(* IEC 61131-3 sources: CodigoPPC/FB da IHM, 6 files *)

(* ---- FC_EpochToString.st ---- *)
// ════════════════════════════════════════════════════════════════════
// FC_EpochToString — Converte UDINT epoch UTC para string legível
// ════════════════════════════════════════════════════════════════════
// Formato: 'DD/MM HH:MM:SS'
// Simplificação: usa SysTimeRtcConvertUtcToLocal + formatação manual
// Se tTimestamp = 0, retorna '-- sem RTC --'
// ════════════════════════════════════════════════════════════════════
FUNCTION FC_EpochToString : STRING(20)
VAR_INPUT
    tEpoch : UDINT;
END_VAR
VAR
    dtLocal     : DT;
    sTemp       : STRING(20);
    nDay        : UINT;
    nMonth      : UINT;
    nHour       : UINT;
    nMin        : UINT;
    nSec        : UINT;
END_VAR

    IF tEpoch = 0 THEN
        FC_EpochToString := '-- sem RTC --';
        RETURN;
    END_IF

    // Converte epoch UDINT para DT (DATE_AND_TIME)
    // DT no CODESYS V3 é segundos desde 01/01/1970 (mesmo que UDINT epoch)
    dtLocal := UDINT_TO_DT(tEpoch);

    // Extrai componentes usando funções padrão do SysTime / Util
    // Nota: a implementação exata depende das libs disponíveis no target.
    // Alternativa simples — usar DT_TO_STRING e truncar:
    sTemp := DT_TO_STRING(dtLocal);

    // DT_TO_STRING retorna formato 'DT#YYYY-MM-DD-HH:MM:SS'
    // Extraímos apenas 'DD/MM HH:MM:SS' (14 chars)
    FC_EpochToString := MID(sTemp, 2, 12);  // DD
    FC_EpochToString := CONCAT(FC_EpochToString, '/');
    FC_EpochToString := CONCAT(FC_EpochToString, MID(sTemp, 2, 9)); // MM
    FC_EpochToString := CONCAT(FC_EpochToString, ' ');
    FC_EpochToString := CONCAT(FC_EpochToString, MID(sTemp, 8, 15)); // HH:MM:SS
END_FUNCTION

(* ---- FC_EventCodeToString.st ---- *)
// ════════════════════════════════════════════════════════════════════
// FC_EventCodeToString — Mensagem legível para E_EventCode (PPC-GD)
// ════════════════════════════════════════════════════════════════════
// Uso: s := FC_EventCodeToString(E_EventCode.CRIT_HARD_LIMIT_15S);
// ════════════════════════════════════════════════════════════════════
FUNCTION FC_EventCodeToString : STRING(80)
VAR_INPUT
    eCode : E_EventCode;
END_VAR

    CASE eCode OF
        // =============================================================
        // NONE
        // =============================================================
        E_EventCode.EVT_NONE:
            FC_EventCodeToString := '';

        // =============================================================
        // INFO (0x1xxx)
        // =============================================================
        // Startup (0x11xx)
        E_EventCode.INFO_STARTUP_BEGIN:
            FC_EventCodeToString := 'Startup: inicio';
        E_EventCode.INFO_SERIAL_COM_OK:
            FC_EventCodeToString := 'Startup: comunicacao serial OK';
        E_EventCode.INFO_RTC_OK:
            FC_EventCodeToString := 'Startup: RTC OK';
        E_EventCode.INFO_INVERTER_COUNT:
            FC_EventCodeToString := 'Startup: quantidade de inversores detectada';
        E_EventCode.INFO_INSTALLED_POWER:
            FC_EventCodeToString := 'Startup: potencia instalada OK';
        E_EventCode.INFO_K1_CONFIRMED:
            FC_EventCodeToString := 'Startup: K1 confirmado';
        E_EventCode.INFO_K2_CONFIRMED:
            FC_EventCodeToString := 'Startup: K2 confirmado';
        E_EventCode.INFO_STARTUP_DONE:
            FC_EventCodeToString := 'Startup: concluido';

        // Medição / Operação (0x12xx)
        E_EventCode.INFO_MEAS_READ_OK:
            FC_EventCodeToString := 'Medidor: leitura OK';
        E_EventCode.INFO_MEAS_DATA_VALID:
            FC_EventCodeToString := 'Medidor: dados validos';
        E_EventCode.INFO_MEAS_RECOVERING:
            FC_EventCodeToString := 'Medicao: recuperando (erros reduzindo)';

        // Escrita inversores (0x13xx)
        E_EventCode.INFO_CH1_WRITE_OK:
    	    FC_EventCodeToString := ' Escrita no canal 01 OK';
    	E_EventCode.INFO_CH2_WRITE_OK:
    	    FC_EventCodeToString := ' Escrita no canal 01 OK';

        // Scheduler (0x15xx)
        E_EventCode.INFO_SPECIAL_DATE_ACTIVE:
            FC_EventCodeToString := 'Scheduler: data especial ativa';
        E_EventCode.INFO_ZERO_GRID_MODE:
            FC_EventCodeToString := 'Scheduler: modo zero grid ativo';

        // Máquina de estados (0x16xx)
        E_EventCode.INFO_CYCLE_COMPLETE:
            FC_EventCodeToString := 'Ciclo: completo';
        E_EventCode.INFO_FAIL_RECOVERY:
            FC_EventCodeToString := 'FAIL: recuperacao automatica';
        E_EventCode.INFO_STATE_CHANGE:
            FC_EventCodeToString := 'Maquina de estados: mudanca de estado';

        // STOP/Reset (0x18xx)
        E_EventCode.INFO_STOP_K2_OPEN_CONFIRMED:
            FC_EventCodeToString := 'STOP: K2 aberto confirmado';
        E_EventCode.INFO_STOP_RESET_APPROVED:
            FC_EventCodeToString := 'STOP: reset aprovado';
        E_EventCode.INFO_STOP_RESET_WAITING:
            FC_EventCodeToString := 'STOP: aguardando reset';

        // =============================================================
        // WARNING (0x2xxx)
        // =============================================================
        // Startup
        E_EventCode.CRIT_TC_POWER_NOT_SET:
            FC_EventCodeToString := 'Startup: TC Power nao configurado';
        E_EventCode.WARN_NO_INVERSORES_COM02:
            FC_EventCodeToString := 'Startup: nenhum inversor no COM2';

        // Medição
        E_EventCode.WARN_MEAS_USING_LAST_VALID:
            FC_EventCodeToString := 'Medicao: usando ultimo valor valido';
        E_EventCode.WARN_MEAS_CROSS_CHECK_PA:
            FC_EventCodeToString := 'Medicao: cross-check Pa falhou';
        E_EventCode.WARN_MEAS_CROSS_CHECK_PB:
            FC_EventCodeToString := 'Medicao: cross-check Pb falhou';
        E_EventCode.WARN_MEAS_CROSS_CHECK_PC:
            FC_EventCodeToString := 'Medicao: cross-check Pc falhou';
        E_EventCode.WARN_MEAS_CROSS_CHECK_PT_SUM:
            FC_EventCodeToString := 'Medicao: cross-check Pt != Pa+Pb+Pc';
        E_EventCode.WARN_MEAS_CROSS_CHECK_PF:
            FC_EventCodeToString := 'Medicao: cross-check PF falhou';
        E_EventCode.WARN_MEAS_ERROR_ISOLATED:
            FC_EventCodeToString := 'Medicao: erro isolado (toleravel)';

        // Comunicação inversores
        E_EventCode.WARN_WRITE_INV_ERROR:
            FC_EventCodeToString := 'Inversores: erro de escrita';
        E_EventCode.WARN_WRITE_INV_TIMEOUT:
            FC_EventCodeToString := 'Inversores: timeout de escrita';

        // Controle
        E_EventCode.WARN_P_ALLOC_SATURATED:
            FC_EventCodeToString := 'Controle: alocacao de P saturada';
        E_EventCode.WARN_Q_LIMITED_BY_SMAX:
            FC_EventCodeToString := 'Controle: Q limitado por Smax';
        E_EventCode.WARN_PF_BELOW_TARGET:
            FC_EventCodeToString := 'Controle: PF abaixo do alvo';
        E_EventCode.WARN_PF_NOT_ACHIEVABLE:
            FC_EventCodeToString := 'Controle: PF nao atingivel';
        E_EventCode.WARN_PI_P_SATURATED:
            FC_EventCodeToString := 'Controle: PI de P saturado';
        E_EventCode.WARN_PI_Q_SATURATED:
            FC_EventCodeToString := 'Controle: PI de Q saturado';
        E_EventCode.WARN_PHASE_LIMITED:
            FC_EventCodeToString := 'Controle: limitado por fase';

        // STOP/reset
        E_EventCode.WARN_STOP_RESET_DENIED:
            FC_EventCodeToString := 'STOP: reset negado';

        // =============================================================
        // ALARM (0x4xxx)
        // =============================================================
        // Medição — Range/Freeze
        E_EventCode.ALARM_MEAS_VOLTAGE_A_RANGE:
            FC_EventCodeToString := 'Medicao: tensao fase A fora de faixa';
        E_EventCode.ALARM_MEAS_VOLTAGE_B_RANGE:
            FC_EventCodeToString := 'Medicao: tensao fase B fora de faixa';
        E_EventCode.ALARM_MEAS_VOLTAGE_C_RANGE:
            FC_EventCodeToString := 'Medicao: tensao fase C fora de faixa';
        E_EventCode.ALARM_MEAS_CURRENT_A_RANGE:
            FC_EventCodeToString := 'Medicao: corrente fase A fora de faixa';
        E_EventCode.ALARM_MEAS_CURRENT_B_RANGE:
            FC_EventCodeToString := 'Medicao: corrente fase B fora de faixa';
        E_EventCode.ALARM_MEAS_CURRENT_C_RANGE:
            FC_EventCodeToString := 'Medicao: corrente fase C fora de faixa';
        E_EventCode.ALARM_MEAS_PT_RANGE:
            FC_EventCodeToString := 'Medicao: Pt fora de faixa';
        E_EventCode.ALARM_MEAS_PA_RANGE:
            FC_EventCodeToString := 'Medicao: Pa fora de faixa';
        E_EventCode.ALARM_MEAS_PB_RANGE:
            FC_EventCodeToString := 'Medicao: Pb fora de faixa';
        E_EventCode.ALARM_MEAS_PC_RANGE:
            FC_EventCodeToString := 'Medicao: Pc fora de faixa';
        E_EventCode.ALARM_MEAS_QT_RANGE:
            FC_EventCodeToString := 'Medicao: Qt fora de faixa';
        E_EventCode.ALARM_MEAS_QA_RANGE:
            FC_EventCodeToString := 'Medicao: Qa fora de faixa';
        E_EventCode.ALARM_MEAS_QB_RANGE:
            FC_EventCodeToString := 'Medicao: Qb fora de faixa';
        E_EventCode.ALARM_MEAS_QC_RANGE:
            FC_EventCodeToString := 'Medicao: Qc fora de faixa';
        E_EventCode.ALARM_MEAS_PFT_RANGE:
            FC_EventCodeToString := 'Medicao: PFt fora de faixa';
        E_EventCode.ALARM_MEAS_PFA_RANGE:
            FC_EventCodeToString := 'Medicao: PFa fora de faixa';
        E_EventCode.ALARM_MEAS_PFB_RANGE:
            FC_EventCodeToString := 'Medicao: PFb fora de faixa';
        E_EventCode.ALARM_MEAS_PFC_RANGE:
            FC_EventCodeToString := 'Medicao: PFc fora de faixa';
        E_EventCode.ALARM_MEAS_FROZEN:
            FC_EventCodeToString := 'Medicao: congelada (frozen)';

        // Comunicação medidor
        E_EventCode.ALARM_MEAS_MODBUS_ERROR:
            FC_EventCodeToString := 'Medidor: erro Modbus';
        E_EventCode.ALARM_MEAS_MODBUS_TIMEOUT:
            FC_EventCodeToString := 'Medidor: timeout';

        // Ciclo / watchdog
        E_EventCode.ALARM_SCAN_OVERRUN:
            FC_EventCodeToString := 'Sistema: scan overrun';

        // Comunicação inversores (canal degradado)
        E_EventCode.ALARM_CH1_MODBUS_ERRO:
            FC_EventCodeToString := 'Canal COM1 >50% falhas';
        E_EventCode.ALARM_CH2_MODBUS_ERRO:
            FC_EventCodeToString := 'Canal COM2 >50% falhas';
        E_EventCode.ALARM_CH1_MODBUS_TIMEOUT:
            FC_EventCodeToString := 'Canal COM1 TIMEOUT < 3x';
        E_EventCode.ALARM_CH2_MODBUS_TIMEOUT:
            FC_EventCodeToString := 'Canal COM2 TIMEOUT < 3x';

        // =============================================================
        // CRITICAL (0x8xxx)
        // =============================================================
        // Startup
        E_EventCode.CRIT_SERIAL_INIT_FAILED:
            FC_EventCodeToString := 'Startup: falha init serial';
        E_EventCode.CRIT_RTC_FAILED:
            FC_EventCodeToString := 'Startup: falha RTC';
        E_EventCode.CRIT_INSTALLED_PWR_ZERO:
            FC_EventCodeToString := 'Startup: potencia instalada = 0';
        E_EventCode.CRIT_K1_TIMEOUT:
            FC_EventCodeToString := 'Startup: timeout K1';

        // Medição
        E_EventCode.CRIT_MEAS_PERSISTENT_FAIL:
            FC_EventCodeToString := 'Medicao: falha persistente';
        E_EventCode.CRIT_MEAS_COM_FAIL:
            FC_EventCodeToString := 'Medidor: falha comunicacao';

        // Comunicação inversores
        E_EventCode.CRIT_INV_CHANNEL_FAIL:
            FC_EventCodeToString := 'Inversores: falha canal comunicacao';

        // Controle
        E_EventCode.CRIT_INSTALLED_POWER_ZERO:
            FC_EventCodeToString := 'Controle: potencia instalada zero';

        // Scheduler
        E_EventCode.CRIT_RTC_READ_FAIL:
            FC_EventCodeToString := 'Scheduler: falha leitura RTC';
        E_EventCode.CRIT_SCHEDULE_INDEX_INVALID:
            FC_EventCodeToString := 'Scheduler: indice invalido';

        // Overrun
        E_EventCode.CRIT_SCAN_OVERRUN:
            FC_EventCodeToString := '3× overruns consecutivos → FAIL';

        // Proteções normativas
        E_EventCode.CRIT_HARDLIMIT_15S:
            FC_EventCodeToString := 'Protecao: HardLimit >15s';
        E_EventCode.CRIT_EXPORT_OVER_LPI_30S:
            FC_EventCodeToString := 'Protecao: Exportacao >LPI >30s';
        E_EventCode.CRIT_MEDIDOR_TIMEOUT_IN_FAIL:
            FC_EventCodeToString := 'Protecao: timeout medidor em FAIL';

        // STOP / Trip
        E_EventCode.CRIT_STOP_ENTRY:
            FC_EventCodeToString := 'STOP: entrada em STOP';
        E_EventCode.CRIT_K2_DID_NOT_OPEN:
            FC_EventCodeToString := 'STOP: K2 nao abriu';
        E_EventCode.CRIT_STATE_CORRUPTION:
            FC_EventCodeToString := 'Sistema: corrupcao de estado';

    ELSE
        FC_EventCodeToString := 'Evento desconhecido';
    END_CASE
END_FUNCTION

(* ---- FC_SeverityToString.st ---- *)
// ════════════════════════════════════════════════════════════════════
// FC_SeverityToString — Extrai severidade do nibble alto de E_EventCode
// ════════════════════════════════════════════════════════════════════
FUNCTION FC_SeverityToString : STRING(8)
VAR_INPUT
    eCode : E_EventCode;
END_VAR
VAR
    nHighNibble : UINT;
END_VAR

    nHighNibble := (TO_UINT(eCode) AND 16#F000);

    CASE nHighNibble OF
        16#1000: FC_SeverityToString := 'INFO';
        16#2000: FC_SeverityToString := 'WARN';
        16#4000: FC_SeverityToString := 'ALARM';
        16#8000: FC_SeverityToString := 'CRIT';
    ELSE
        FC_SeverityToString := '???';
    END_CASE
END_FUNCTION

(* ---- FC_UIntToHex16Sharp.st ---- *)
// ════════════════════════════════════════════════════════════════════
// FC_UIntToHex16Sharp — Formata UINT como '16#XXXX' (4 nibbles)
// Ex.: 16#8700 -> '16#8700'
// tentar usar UINT_TO_HEXSTR se o CODESYS aceitar
// ════════════════════════════════════════════════════════════════════
FUNCTION FC_UIntToHex16Sharp : STRING(7)
VAR_INPUT
    uValue : UINT;
END_VAR
VAR
    aHex   : STRING(16) := '0123456789ABCDEF';
    n0, n1, n2, n3 : UINT;
    sOut : STRING(7);
END_VAR

    n3 := (uValue AND 16#000F);
    n2 := (SHR(uValue, 4)  AND 16#000F);
    n1 := (SHR(uValue, 8)  AND 16#000F);
    n0 := (SHR(uValue, 12) AND 16#000F);

    // Monta '16#' + 4 dígitos
    sOut := '16#';
    sOut := CONCAT(sOut, MID(aHex, n0 + 1, 1));
    sOut := CONCAT(sOut, MID(aHex, n1 + 1, 1));
    sOut := CONCAT(sOut, MID(aHex, n2 + 1, 1));
    sOut := CONCAT(sOut, MID(aHex, n3 + 1, 1));

    FC_UIntToHex16Sharp := sOut;
END_FUNCTION

(* ---- FB_EventDisplay.st ---- *)
// ════════════════════════════════════════════════════════════════════
// FB_EventDisplay — Prepara eventos do ring buffer para exibição na IHM
// ════════════════════════════════════════════════════════════════════
// A IHM não navega o ring buffer diretamente. Este FB expõe
// N linhas "flat" prontas para bind em Text Fields.
//
// Suporta paginação: nPageOffset controla qual "página" exibir.
//   Página 0 = eventos mais recentes
//   Página 1 = próximos DISPLAY_LINES eventos, etc.
//
// Chamado sob demanda (quando operador abre a tela de histórico),
// NÃO a cada ciclo.
// ════════════════════════════════════════════════════════════════════
FUNCTION_BLOCK FB_EventDisplay

VAR_INPUT
    pEventLog       : REFERENCE TO FB_EventLog;     // Referência ao ring buffer
    bRefresh        : BOOL;                         // Pulso = atualiza dados
    nPageOffset     : UINT := 0;                    // Página (0 = mais recente)
END_VAR

VAR_OUTPUT
    nTotalEvents    : UINT;                         // Total de eventos no buffer
    nTotalPages     : UINT;                         // Total de páginas disponíveis
    nCurrentPage    : UINT;                         // Página atual (0-based)
END_VAR

VAR CONSTANT
    DISPLAY_LINES   : UINT := 10;                   // Linhas visíveis na tela
END_VAR

VAR
    // ── Dados "flat" para a IHM (cada linha = 1 evento) ──
	(*
	ST_EventOutput
    asTimestamp      : STRING(20);   // 'DD/MM HH:MM:SS'
    asMessage        : STRING(60);   // Mensagem legível
    asParam1         : STRING(12);   // Valor contexto 1
    asParam2         : STRING(12);   // Valor contexto 2
    asSeverity       : STRING(8);    // 'INFO'/'WARN'/'ALARM'/'CRIT'
    asRaised         : STRING(5);    // 'RAISE' / 'CLEAR'
    abLineValid      : BOOL;         // TRUE = linha tem dados
	asCodeHex        : STRING(8);    // ex: '16#8700'
	*)

    Display     	: ARRAY[0..9] OF ST_EventOutput;

    // Auxiliares
    i               : UINT;
    nStartIdx       : UINT;
    stEvt           : ST_EventEntry;
    bOK             : BOOL;
    rTrigRefresh    : R_TRIG;
END_VAR

    // ════════════════════════════════════════════════════════════════════
    // Corpo do FB_EventDisplay — executa quando bRefresh tem borda de subida
    // ════════════════════════════════════════════════════════════════════
    rTrigRefresh(CLK := bRefresh);

    IF rTrigRefresh.Q THEN

        // Total de eventos e páginas
        nTotalEvents := pEventLog.nCount;
        IF nTotalEvents > 0 THEN
            nTotalPages := ((nTotalEvents - 1) / DISPLAY_LINES) + 1;
        ELSE
            nTotalPages := 0;
        END_IF

        // Clamp página
        IF nPageOffset >= nTotalPages THEN
            nPageOffset := 0;
        END_IF
        nCurrentPage := nPageOffset;

        // Índice inicial no ring buffer (reverso)
        nStartIdx := nPageOffset * DISPLAY_LINES;

        // Preencher linhas
        FOR i := 0 TO (DISPLAY_LINES - 1) DO

            bOK := pEventLog.GetEvent(
                nReverseIndex := nStartIdx + i,
                stOut => stEvt
            );

            IF bOK THEN
                Display[i].abLineValid := TRUE;

                // Timestamp → string legível
                Display[i].asTimestamp := FC_EpochToString(stEvt.tTimestamp);

                // Código → mensagem
                Display[i].asMessage := FC_EventCodeToString(stEvt.eCode);

                // Severidade (extraída do nibble alto do código)
                Display[i].asSeverity := FC_SeverityToString(stEvt.eCode);

                // Raise/Clear
                IF stEvt.bRaised THEN
                    Display[i].asRaised := 'RAISE';
                ELSE
                    Display[i].asRaised := 'CLEAR';
                END_IF

                // Parâmetros numéricos formatados
                Display[i].asParam1 := REAL_TO_STRING(stEvt.rParam1);
                Display[i].asParam2 := REAL_TO_STRING(stEvt.rParam2);
    			Display[i].asCodeHex := FC_UIntToHex16Sharp(TO_UINT(stEvt.eCode));
            ELSE
                // Linha vazia
                Display[i].abLineValid  := FALSE;
                Display[i].asTimestamp  := '';
                Display[i].asMessage    := '';
                Display[i].asSeverity   := '';
                Display[i].asRaised     := '';
                Display[i].asParam1     := '';
                Display[i].asParam2		:= '';
    			Display[i].asCodeHex	:= '';
            END_IF

        END_FOR

    END_IF
END_FUNCTION_BLOCK

(* ---- TaskIHM.st ---- *)
PROGRAM TaskIHM
VAR
	    fbEventDisplay  		: FB_EventDisplay;			// prepara dados para a IHM

	// ══════════════════════════════════════════════════════════
	// Variáveis manipuladas pela IHM
	// ══════════════════════════════════════════════════════════
 	HMI_bRefresh    		: BOOL;     // Botão "Refresh" na IHM (pulso)
    HMI_nPage       		: UINT;     // Página atual (0 = mais recente)

END_VAR

    // Chama o FB de display todo ciclo (ele só recalcula quando HMI_bRefresh der pulso)
    fbEventDisplay(
        pEventLog   := GVL_Main.fbEventLog,     // referência ao ring buffer
        bRefresh    := HMI_bRefresh,   			// pulso da IHM
        nPageOffset := HMI_nPage       			// página selecionada
    );
END_PROGRAM
